{attribute 'qualified_only'}
VAR_GLOBAL

    (* color inputs for each machine *)
    colorMachine : ARRAY[1..10] OF INT;

END_VAR

(* stored: Version 1.1.0.1
   GVL GVL: Id {aa48bf9c-aed2-468f-8ef2-bcf9df62a85b} *)
